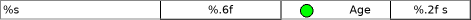
VISUALIZATION VISU_AlpacaGetLreal  // 471x20
VAR_IN_OUT
	stInstance : ST_AlpacaGetLreal;
END_VAR
    Rectangle (160,0 121x20), "%.6f", text variable: stInstance.lrValue
    Rectangle (0,0 161x20), "%s", text variable: stInstance.sName
    Ellipse (300,4 13x13), colour toggle: stInstance.eStatusCode <> E_AlpacaStatusCode.OK
    Rectangle (390,0 81x20), "%.2f s", text variable: stInstance.rAge
    Label (340,0 41x20), "Age"
END_VISUALIZATION

(* stored: Version 1.1.0.1, ProductVersion 3.1.4024.12
   Visu VISU_AlpacaGetLreal: Id {a7ae4a94-e0a1-4b20-a0da-58a1376adefa} *)
